INTERFACE I_Skill_Roboter

METHOD M_Reset : BOOL
VAR_INPUT
END_VAR
END_METHOD

METHOD M_Start : BOOL
VAR_INPUT
END_VAR
END_METHOD

METHOD M_Stop : BOOL
VAR_INPUT
END_VAR
END_METHOD

PROPERTY P_RobotParam : sRoboterProzessVariablen
SET
END_SET
END_PROPERTY

PROPERTY P_State : eSkillState
GET
END_GET
END_PROPERTY

END_INTERFACE

(* stored: Version 1.1.0.1
   Itf I_Skill_Roboter: Id {25ddb587-d49a-4ab5-8d90-3b97fd134ecd}
   Method M_Reset: Id {5abbd829-ae4b-4033-9c7c-a8e9718f05af}
   Method M_Start: Id {60d386b6-acdc-4f5b-a440-ee35cb2a066c}
   Method M_Stop: Id {a2533550-c461-4226-9eb6-58f5b281cdae}
   Property P_RobotParam: Id {e54f29bf-49d9-404d-a7ec-63c18cdf5712}
   Set Set: Id {8f450706-785d-4a6e-aaca-766c387026dd}
   Property P_State: Id {71a4ac71-288b-425c-80e9-8937cbbaa14d}
   Get Get: Id {f97b7deb-80ff-4671-ab0c-6da64dba1568} *)
